% RSLogix 500 project sti_1000ms_live.RSS, saved by version 8.30.00.16 %
PROJECT "UNTITLED"    % processor: Bul.1763 MicroLogix 1100 Series B %

PROGRAM FILES
  LAD 2   5 rungs
  LAD 3   2 rungs

DATA FILES
  O0 OUTPUT  4 elements
  I1 INPUT  6 elements
  S2 STATUS  66 elements
  B3 BINARY  1 elements
  T4 TIMER  1 elements
  C5 COUNTER  1 elements
  R6 CONTROL  1 elements
  N7 INTEGER  20 elements
  F8 FLOAT  1 elements
  N9 DELTATIMES  256 elements

LADDER 2
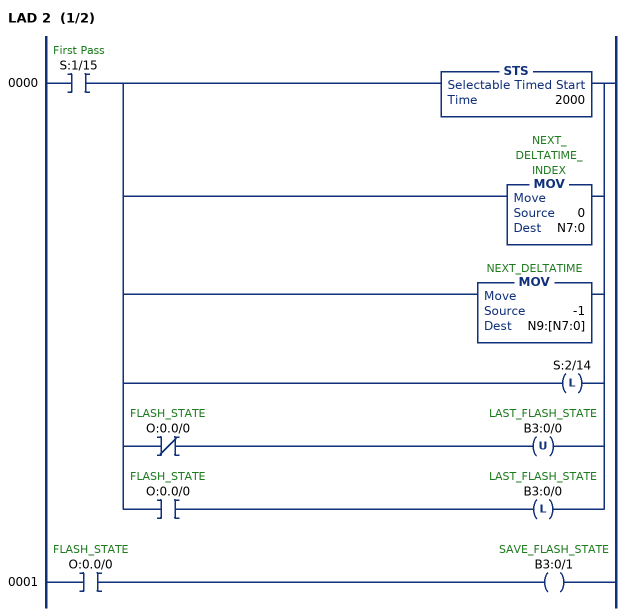
% Rung: 0 %
SOR XIC S:1/15 BST STS 2000 NXB MOV 0 N7:0 NXB MOV -1 N9:[N7:0] NXB OTL S:2/14 NXB XIO O:0.0/0 OTU B3:0/0 NXB XIC O:0.0/0 OTL B3:0/0 BND EOR
%   S:1/15  "First Pass" %
%   N7:0  NEXT_DELTATIME_INDEX %
%   N9:[N7:0]  NEXT_DELTATIME %
%   O:0.0/0  FLASH_STATE %
%   B3:0/0  LAST_FLASH_STATE %
% Rung: 1 %
SOR XIC O:0.0/0 OTE B3:0/1 EOR
%   O:0.0/0  FLASH_STATE %
%   B3:0/1  SAVE_FLASH_STATE %

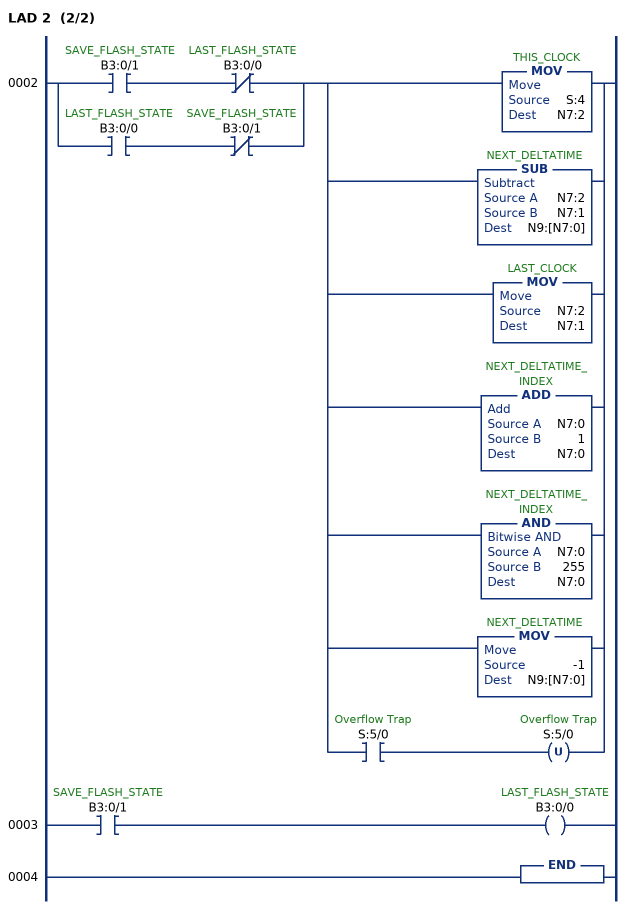
% Rung: 2 %
SOR BST XIC B3:0/1 XIO B3:0/0 NXB XIC B3:0/0 XIO B3:0/1 BND BST MOV S:4 N7:2 NXB SUB N7:2 N7:1 N9:[N7:0] NXB MOV N7:2 N7:1 NXB ADD N7:0 1 N7:0 NXB AND N7:0 255 N7:0 NXB MOV -1 N9:[N7:0] NXB XIC S:5/0 OTU S:5/0 BND EOR
%   B3:0/1  SAVE_FLASH_STATE %
%   B3:0/0  LAST_FLASH_STATE %
%   S:4  "Time Base" %
%   N7:2  THIS_CLOCK %
%   N7:1  LAST_CLOCK %
%   N9:[N7:0]  NEXT_DELTATIME %
%   N7:0  NEXT_DELTATIME_INDEX %
%   S:5/0  "Overflow Trap" %
% Rung: 3 %
SOR XIC B3:0/1 OTE B3:0/0 EOR
%   B3:0/1  SAVE_FLASH_STATE %
%   B3:0/0  LAST_FLASH_STATE %
% Rung: 4 %
SOR END EOR

LADDER 3
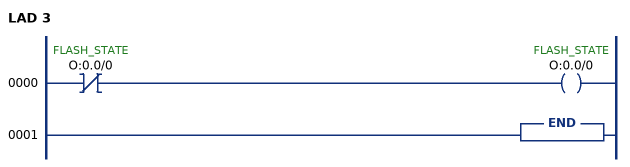
% Rung: 0 %
SOR XIO O:0.0/0 OTE O:0.0/0 EOR
%   O:0.0/0  FLASH_STATE %
% Rung: 1 %
SOR END EOR

OTHER DOCUMENTED ADDRESSES
  I:0.0/[N7:1]  TANK_BY_INDEX_STATE
  RTC:0.SEC/1  LAMP_FLASH_RTC_BIT01

DATA TABLE (non-zero values as saved)
DATA B3
% B3:0 % 0X0003
DATA N7
% N7:0 % 7 17696 17696 0 0 0 0 0 0 0
DATA N9
% N9:0 % 20000 20006 20001 20002 20001 19999 20002 -1 19999 20004
% N9:10 % 20001 20007 20001 20000 20003 20004 19998 20002 20006 20008
% N9:20 % 19999 20000 20003 20000 20001 20005 19999 20001 20006 19997
% N9:30 % 20006 20000 20008 19995 20009 20002 20001 20001 19998 20004
% N9:40 % 20002 20005 20003 20004 20000 20003 20000 20002 20000 20004
% N9:50 % 20004 19997 20006 20003 20001 20001 20004 20001 19999 20005
% N9:60 % 20001 20002 20005 20003 20001 19997 20004 20004 20003 20001
% N9:70 % 20000 20011 20004 20002 19997 20001 20007 19999 20001 20003
% N9:80 % 19999 20005 20000 20004 19999 20005 20001 20002 20002 20002
% N9:90 % 20001 20004 19999 20005 20002 20004 19997 20006 20003 19999
% N9:100 % 20002 20001 20002 20004 20002 20004 19999 20006 19998 20007
% N9:110 % 19997 20005 20004 20001 20000 20003 20004 20002 19999 20006
% N9:120 % 19998 20003 20000 20009 20001 20003 19999 20004 20004 20003
% N9:130 % 19997 20005 20004 20001 20000 20005 20001 19999 20006 20000
% N9:140 % 20005 19996 20002 20007 19998 20007 19997 20006 20002 20001
% N9:150 % 20006 19998 20005 19996 20008 20003 19996 20006 20002 20003
% N9:160 % 20002 20000 20000 20007 20003 19997 20004 20005 20002 19999
% N9:170 % 20004 20002 19999 20013 19992 20013 19998 20006 19995 20009
% N9:180 % 19994 20006 19999 20003 20003 20000 20004 20002 19999 20004
% N9:190 % 19999 20002 20007 20003 19997 20005 20004 19999 20004 20001
% N9:200 % 20001 20003 20006 20006 19996 19999 20001 20005 20002 20001
% N9:210 % 20006 20001 20002 19998 20003 20004 20001 20002 20004 20000
% N9:220 % 20004 20003 20004 20000 20002 20004 20004 19998 20002 20002
% N9:230 % 20006 20002 20000 19999 20005 19998 20006 20002 20002 20002
% N9:240 % 20003 20001 20000 20005 19999 20003 20005 20001 19999 20007
% N9:250 % 20002 20001 19999 20007 20002 20001
